FUNCTION_BLOCK ABSTRACT FB_WorkerDefGrid EXTENDS FB_Worker
VAR_OUTPUT
  bError            : BOOL;                           // an error is active
  nError            : UDINT;                          // error code if error active, =0 else
END_VAR
VAR
  // config
  _pMsgConfigExt    : POINTER TO ST_MSG_CONFIG;       // external message config (puc message interface)
  _fPrintResolution : LREAL := 1;                     // print(head) resolution in [dpi]
  _fSubPxResolution : LREAL := 1;                     // SubPixel resolution [SubPx], resolution factor (fI_PrintResolution*fI_SubPxResolution=>Output resolution
  _name             : STRING;                         // Worker name
  _sVisuName        : STRING := 'VISU_WorkerDefGrid'; // Worker visu instance name
  _pEcSrc           : POINTER TO T_ErrSrc;            // Error source definition

  // job
  _bJobActive       : BOOL;                           // a job is active
  // ct
  _bAttached        : BOOL;                           // one ct is attached
  _pAttachedCt      : POINTER TO FB_ContainerDefGrid; // currently attached container (Head)
  _pNewAttached     : POINTER TO FB_ContainerDefGrid; // last attached container (as return value of Attach() (Tail))
  _bSupportParallelCT : BOOL := FALSE;                // support for parallel CTs (else avoid attach while one connected).
  _nAttachedCTs     : UDINT;                          // Number of currently attached CTs
  _pAttachedCTList  : ARRAY[nLowerIndexCTList..nUpperIndexCTList] OF POINTER TO FB_ContainerDefGrid;
  // position control
  fCtPosition       : LREAL;     // Container position relative to worker position
  _bForceRelease    : BOOL;                           // Manually force a ct release

  // view
  nGridRowStart, nGridColStart: UDINT := 0;
END_VAR
VAR_STAT
  // static variables, SAME for ALL Workers
  _pCTM             : POINTER TO FB_CTManagerDefGrid;             // "Global" Container Manager
  _fCtSecurityReleasePos : LREAL := 0;                // [SubPx] position where to release current ct at last (security release)
END_VAR
VAR PERSISTENT
  _fWorkerPosition  : LREAL;                          // [m] worker distance to X0 (position from X0) (CT creation X0 and domain)
END_VAR
VAR CONSTANT
  fC_MaxSheetLengthExtension : LREAL := 0.30;         // Max. distance after given ImageLength to do security release of CT
  // list size
  nLowerIndexCTList : UDINT := 1;
  nUpperIndexCTList : UDINT := 4; 
END_VAR

(*
  Generic abort implementation of DefGrid CT.
*)
METHOD Abort
VAR_INPUT
  iCT       : I_CT;
  sReason   : STRING;
END_VAR
VAR
  _pCt   : POINTER TO FB_ContainerDefGrid;
  eStep     : E_DeformationStep;
END_VAR
IF iCT = 0 AND _pAttachedCt <> 0 THEN             // no ct given and check if one is attached 
  _pCt := _pAttachedCt;
ELSIF getCtInst(iCT:=iCT, pCT=>_pCt) = 0 THEN     // get specific container from given interface
  RETURN; 
END_IF

IF _pCt = 0 THEN RETURN; END_IF
  
// abort CT
  // Do generic known aborts on CT
  // - Deformation
  _pCt^.getDeformationStatus(eDStep=>eStep);
  IF eStep >= E_DeformationStep.nothing THEN
    _pCt^.AbortDeformation(sReason:=sReason, Src:=_pEcSrc^, bHideLog:=FALSE);
  
END_IF
END_METHOD

METHOD PROTECTED  Attach : BOOL
VAR_INPUT
  iCT       : I_CT;            (*container at triggered event position*)
END_VAR
VAR
  i : UDINT;
END_VAR
Attach := FALSE;

IF iCT = 0 THEN
  LogError(Msg:='attach failed -> not ct given');
  
ELSIF bWorkerEnable THEN  // worker enabled
  
  IF getCtInst(iCT:=iCT, pCT=>_pNewAttached) <> 0 THEN    // get specific container
    // add to list ()
    IF push(pNewCT:=_pNewAttached) THEN 
      LogLvl(Lvl:=E_LogSeverity.Debug, Msg:=F_Concat4('Attach CT[', TO_STRING(_nAttachedCTs), ']: ', _pNewAttached^.print(0)));
      Attach:=TRUE;                                 // attach new
    END_IF
  ELSE
    LogError(Msg:='attach failed: could not get CT instance');
  END_IF

ELSIF NOT bWorkerEnable AND _nAttachedCTs > 0 THEN // disabled and already a CT attached
  // force release all attached CT, and ignore attach
  LogLvl(Lvl:=E_LogSeverity.Debug, Msg:='Worker disabled flush list of all attached CT');
  WHILE _nAttachedCTs > 0 DO
    Release(iCT:=_pAttachedCt^);
	END_WHILE

ELSIF NOT bWorkerEnable AND _pAttachedCt = 0 THEN  
  ;   // nothing to do, ignore attach

ELSE      // unspecified (error)case just log it
  LogError(Msg:='not tracked case');
END_IF


// ok to attach
END_METHOD

{attribute 'monitoring':='call'}
PROPERTY bAttached : BOOL
GET
bAttached := _bAttached;
END_GET
END_PROPERTY

{attribute 'monitoring':='call'}
PROPERTY fPosition : LREAL
GET
fPosition := _fWorkerPosition;
END_GET
SET
_fWorkerPosition := fPosition;  // [m] save position
END_SET
END_PROPERTY

(*
  Get specific container from interface.
  Returns specific container in return value and output parameter.
*)
METHOD INTERNAL getCtInst : POINTER TO FB_ContainerDefGrid
VAR_INPUT
  iCT              : I_CT;                         (*container at triggered event position*)
END_VAR
VAR_OUTPUT
  pCT              : POINTER TO FB_ContainerDefGrid;
END_VAR
IF NOT bInitialized THEN RETURN; END_IF
IF _pCTM = 0 THEN RETURN; END_IF

pCT := 0;
getCtInst := _pCTM^.GetContainerInstance(iCT);   // get real ct fb inst
IF getCtInst <> 0 THEN
  pCT := getCtInst;   // OK all good
ELSE
  LogError(Msg:='specific container not found');
END_IF
END_METHOD

(*
  Get relative position to this worker (relative to track position)
*)
METHOD getPosRelToAttach : DINT
VAR_INPUT
  iCT : I_CT;
END_VAR
// relative position to X0 - tracking offset of this worker
getPosRelToAttach := _iCTTracker.getPosRel(iCT:=iCT)-_nTrackOffset;
END_METHOD

METHOD Init
VAR_INPUT
  pMsgConfig : POINTER TO ST_MSG_CONFIG;         // message config
  fPrintResolution : LREAL := 1;                 // print(head) resolution in [dpi]
  fSubPxResolution : LREAL := 1;                 // SubPixel resolution [SubPx], resolution factor (fI_PrintResolution*fI_SubPxResolution=>Output resolution)
  bParallelCT : BOOL;                            // Support parallel processing of CTs
END_VAR
VAR

END_VAR
_bAttached := 0;
_pAttachedCt := 0;
_nAttachedCTs := 0;

IF _pCTM = 0 THEN LogError(Msg:='Init: invalid parameter'); RETURN; END_IF

// save config
_pMsgConfigExt := pMsgConfig;
_fPrintResolution := fPrintResolution;
_fSubPxResolution := fSubPxResolution;
_fCtSecurityReleasePos := 0;
_bSupportParallelCT := bParallelCT;

setName('');

// init error source reference
_pEcSrc := ErrorCodes.fbErrCodeMngr.registerErrSource(
  nLocId := 0,
  aInstPath := InstanceName,
  aLocDescr := _name
);
IF _pEcSrc = 0 THEN LogError('could not register error source'); END_IF

bInitialized := TRUE;
END_METHOD

METHOD ABSTRACT mJobStart
VAR_INPUT
	sJobDef	: CalmarCompPrint.I_JobDefinition;
END_VAR
END_METHOD

METHOD ABSTRACT mJobStop
VAR_INPUT
	sStatus	: CalmarCompPrint.I_JobStatus;
END_VAR
END_METHOD

PROPERTY pCTM : POINTER TO FB_CTManagerDefGrid
GET
pCTM := _pCTM;
END_GET
SET
_pCTM := pCTM;
END_SET
END_PROPERTY

METHOD PRIVATE pull : BOOL
VAR_INPUT
  pRemCT : POINTER TO FB_ContainerDefGrid;
END_VAR
VAR_OUTPUT
  nRemIndex : DINT := 0;
END_VAR
VAR
  i                : DINT;
  Index            : DINT;
  LowerIndex       : DINT := 1;
END_VAR
IF _nAttachedCTs = 0 THEN LogError('Release: but no CT is attached'); RETURN; END_IF

// -- find if ct is in attached list
Index := -1;
FOR i:= TO_DINT(nLowerIndexCTList) TO TO_DINT(nLowerIndexCTList + _nAttachedCTs - 1) DO
  IF _pAttachedCTList[i] = pRemCT THEN
    Index := i;
    EXIT;     // found
  END_IF
END_FOR
IF Index = -1 THEN LogError('Release: ct inst not found in list'); RETURN; END_IF

// do stop CT callback if removing first
IF Index = TO_DINT(nLowerIndexCTList) THEN StopCT(pCtDefGrid:=pRemCT); END_IF

// compress list
IF Index >= TO_DINT(nLowerIndexCTList) AND Index < TO_DINT(nUpperIndexCTList) THEN
  MEMMOVE(              // shift all above entries down
    destAddr := ADR( _pAttachedCTList[Index] ), 
    srcAddr  := ADR( _pAttachedCTList[Index + 1] ), 
    n        := DINT_TO_UDINT(SIZEOF(_pAttachedCTList[LowerIndex]) * (UDINT_TO_DINT(_nAttachedCTs) - Index - 1 + LowerIndex))
  );
  _pAttachedCTList[nUpperIndexCTList] := 0;   // erase last(compressed) list entry
END_IF
_pAttachedCTList[_nAttachedCTs] := 0;   // erase last element

// remove
_nAttachedCTs := _nAttachedCTs - 1;   // remove one element

IF _nAttachedCTs > 0 THEN 
  // Start new HEAD
  _pAttachedCt := _pAttachedCTList[1];
  _bAttached := TRUE;
  StartCT(pCtDefGrid:=_pAttachedCt);
ELSE
  // CT list empty (no ct attached)
  _pAttachedCt := 0;
  _bAttached := 0;
END_IF

nRemIndex := Index;
pull := TRUE;
END_METHOD

METHOD PRIVATE push : BOOL
VAR_INPUT
  pNewCT : POINTER TO FB_ContainerDefGrid;
END_VAR
// checks
// - valid param
IF pNewCT = 0 THEN LogError('push: invalid pointer'); RETURN; END_IF
// - list full
IF _nAttachedCTs >= nUpperIndexCTList THEN  // list overflow no free element for processing
  LogError('Worker processing list full, ignore new CT');
  Abort(iCT:=pNewCT^, sReason:='attach failed: too many attached');  // abort new CT (no release because not yet attached)
  RETURN;
END_IF
// - only one CT allowed
IF _nAttachedCTs > 0 AND NOT _bSupportParallelCT THEN
  LogError(Msg:='another container already attached -> ignore new (set error)');
  Abort(iCT:=pNewCt^, sReason:='attach failed: no parallel support');  // abort new CT
END_IF

// add to list
_nAttachedCTs := _nAttachedCTs + 1;
_pAttachedCTList[_nAttachedCTs] := pNewCT;

// apply head
IF _nAttachedCTs = 1 THEN
  // set HEAD
  _pAttachedCt := _pAttachedCTList[nLowerIndexCTList];  
  _bAttached := TRUE;
  
  // start callback on HEAD
  StartCT(pCtDefGrid:=_pAttachedCt);
END_IF

push := TRUE;
END_METHOD

(*
  Release CT from Worker.
  :return: TRUE if CT was released, FALSE if no CT was registered 
*)
METHOD Release : BOOL
VAR_INPUT
  iCT              : I_CT;                         (*container at triggered event position*)
END_VAR
VAR
  nIdx             : DINT;
  pCT              : POINTER TO FB_ContainerDefGrid;
END_VAR
// remove CT -----------------------------------------------------
// -- get real instance
pCT := getCtInst(iCT:=iCT);
IF pCT = 0 THEN LogError('Release: could not find ct instance'); RETURN; END_IF

// remove and release CT
IF pull(pRemCT:=pCT, nRemIndex=>nIdx) THEN
  LogLvl(Lvl:=E_LogSeverity.Debug, Msg:=F_Concat4('Release CT[', TO_STRING(nIdx), '] ', pCt^.print(0)));
  Release := TRUE;  
END_IF
END_METHOD

METHOD PRIVATE setName : BOOL
VAR_INPUT
  sName : STRING;
END_VAR
VAR
  nIdx : INT;
  bDone : BOOL;
END_VAR
IF sName = '' THEN
  // generate worker name
  _name := THIS^.InstanceName;
  WHILE NOT bDone DO
    nIdx := FIND(_name, '.');
    IF nIdx = 0 THEN bDone := TRUE; EXIT; 
    ELSE
      _name := RIGHT(_name,LEN(_name)-nIdx);
    END_IF 
  END_WHILE
ELSE
  _name := sName;  
END_IF
END_METHOD

METHOD PROTECTED StartCT
VAR_INPUT
 pCtDefGrid   : POINTER TO FB_ContainerDefGrid;
END_VAR
(* Override specific implementation in child class *)
END_METHOD

METHOD PROTECTED StopCT
VAR_INPUT
 pCtDefGrid   : POINTER TO FB_ContainerDefGrid;
END_VAR
(* Override specific implementation in child class *)
END_METHOD

METHOD  work
VAR
  i : UDINT;
  pCt : POINTER TO FB_ContainerDefGrid;
END_VAR
// set tracking offset
_nTrackOffset := F_MeterToSubPixel(fPosMeter:=fPosition, fResoSubPx:=_fPrintResolution*_fSubPxResolution);  // [pos domain] save position

//Work only with attached container
IF _nAttachedCTs = 0 THEN RETURN; END_IF
  
FOR i:=nLowerIndexCTList TO nLowerIndexCTList + _nAttachedCTs - 1 DO
  pCt := _pAttachedCTList[i];

  // update CT position
  fCtPosition := getPosRelToAttach(iCT:=pCt);
  
  // release CT (manually)
  IF _bForceRelease THEN
    //Abort(iCT:=pCt^, sReason:='Manually realease CT');
    LogWarning(F_Concat2('Manually realease CT Id=', TO_STRING(pCt^.pCT^.iId)));
    Release(iCT:=pCt^);

  // security release 
  ELSIF _fCtSecurityReleasePos > 0 AND (fCtPosition > _fCtSecurityReleasePos) THEN
    //Abort(iCT:=pCt^, sReason:=F_Concat2('Security released CT Id=', TO_STRING(pCt^.pCT^.iId)));
    LogError(F_Concat2('Security released CT Id=', TO_STRING(pCt^.pCT^.iId)));
    Release(iCT:=pCt^);
  END_IF

END_FOR
END_METHOD

END_FUNCTION_BLOCK

(* stored: Version 1.1.0.1, ProductVersion 3.1.4024.11
   POU FB_WorkerDefGrid: Id {ec3f04b6-f22a-4a73-9fd6-d551c3304c16}, SpecialFunc None
   Folder CTList: Id {8b3e6e49-2ffc-4cad-96ea-0e5e1e9c12fb}
   Folder I_PrintStatusClient: Id {522437a3-298d-4e2e-9ebe-709d3e172129}
   Method Abort: Id {f8718905-c76d-49a9-949e-6da2bac3e031}
   Method Attach: Id {6e998c00-d198-4ad0-b5d5-92dbb9b30114}
   Property bAttached: Id {2e8c8130-f685-40b1-adbf-abe31d58117b}
   Get Get: Id {02ef1e0c-6e3d-4b78-a33e-9b7da2b704a6}
   Property fPosition: Id {9e6d5cd4-bcef-45e7-9eee-8ae16a558520}
   Get Get: Id {1b62f39a-72fb-46df-8d2d-82b64e6e95db}
   Set Set: Id {c5124a02-dd31-4a8c-a934-986e277cf211}
   Method getCtInst: Id {97cf106b-4be9-4376-a613-0f240f49b306}
   Method getPosRelToAttach: Id {bbe24514-8a31-4018-8f0f-1e46c4dca809}
   Method Init: Id {9892d34e-806e-432a-b876-226a7f31ec11}
   Method mJobStart: Id {2edcddcb-d5cc-4bb1-81a9-c6fb86b8259f}
   Method mJobStop: Id {440aa514-bfaa-418c-8033-255390b9e116}
   Property pCTM: Id {94eae062-0ad0-4489-9e76-230fab325e73}
   Get Get: Id {9a767bc1-2f28-4654-9da9-7590f4296c7f}
   Set Set: Id {73378995-26ab-4925-ad9b-1f6205314d3e}
   Method pull: Id {5e0f29fc-a1aa-456a-98f0-78a2b334b213}
   Method push: Id {c3c7aaec-1980-4a48-a4a7-8390a6d54bae}
   Method Release: Id {0d710157-0566-4311-84ad-ccf34b31ce11}
   Method setName: Id {66618658-df51-457a-bb97-2f422320d543}
   Method StartCT: Id {28400007-7a5d-4fce-a93d-03d5259530e3}
   Method StopCT: Id {cf4cd522-5869-4bb8-853b-bccf0021d001}
   Method work: Id {3d2d038f-b3d5-4af3-8623-edc2cf824dd4} *)
